{attribute 'qualified_only'}
VAR_GLOBAL
END_VAR

(* stored: Version 1.1.0.1, ProductVersion 3.1.4024.11
   GVL GVL_Bus: Id {b62cb967-bd7a-4cae-98f9-001cc27e529c} *)
